TYPE ST_PD4_HW :
STRUCT
	StatusWord 				AT %I* : UINT; 
	OperationModeDisplay 	AT %I* : SINT;
	ActualPosition 			AT %I* : DINT;
	ActualVelocity 			AT %I* : INT;
	
	
	ControlWord 	AT %Q* : UINT;
	HomingMethod 	AT %Q* : USINT;
	TargetVelocity 	AT %Q* : INT;
	ProfileVelocity AT %Q* : UDINT;
	Accel 			AT %Q* : UDINT;				
	Decel 			AT %Q* : UDINT;				
	SubmodeSelect	AT %Q* : UDINT;	
	OperationMode 	AT %Q* : SINT;	
	TargetPosition 	AT %Q* : DINT;		
	Polarity 		AT %Q* : USINT;		
END_STRUCT
END_TYPE

(* stored: Version 1.1.0.1, ProductVersion 3.1.4024.12
   DUT ST_PD4_HW: Id {f06f883a-37bf-0d7e-21ea-82ba45b80149} *)
